(* IEC 61131-3 sources: repolevel_ST_code_completion/output/0127完整版本_带planner/repoeval_elevator/readful_result_no_provide, 4 files *)

(* ---- F_DetectCurrentFloor.st ---- *)
IF FloorSensor0 THEN
	F_DetectCurrentFloor := 0;
ELSIF FloorSensor1 THEN
	F_DetectCurrentFloor := 1;
ELSIF FloorSensor2 THEN
	F_DetectCurrentFloor := 2;
ELSIF FloorSensor3 THEN
	F_DetectCurrentFloor := 3;
ELSE
	F_DetectCurrentFloor := CurrentFloor;
END_IF;
RETURN;
END_FUNCTION

(* ---- F_UpdateDoorAnimation.st ---- *)
VAR
	nNewAni			:	DINT;		// 新的动画值
END_VAR

nNewAni := nCurrentAni;

// 开门动画（增加动画值）
IF bOpenDoor AND nNewAni < nMaxAni THEN
	nNewAni := nNewAni + 1;
END_IF

// 关门动画（减少动画值）
IF bCloseDoor AND nNewAni > 0 THEN
	nNewAni := nNewAni - 1;
END_IF

// 楼层呼叫动画（增加动画值）
IF bCallFloor AND nNewAni < nMaxAni THEN
	nNewAni := nNewAni + 1;
END_IF

// 保持动画值不变
IF NOT bCallFloor AND NOT bOpenDoor AND NOT bCloseDoor THEN
	nNewAni := nCurrentAni;
END_IF

F_UpdateDoorAnimation := nNewAni;
END_FUNCTION

(* ---- FB_ElevatorDoorController.st ---- *)
VAR
	fbDoorTimer			:	TON;		// 开门延时定时器
	fbCloseDoorTimer	:	TON;		// 关门延时定时器
	nState				:	INT;		// 状态机
	bEmergencyStop		:	BOOL;		// 紧急停止信号
END_VAR

CASE nState OF
	0: // 空闲状态
		bOpenDoor := FALSE;
		bCloseDoor := FALSE;
		bDoorOpen := FALSE;
		bDoorReady := TRUE;

		IF bArrivedAtTarget THEN
			nState := 1; // 开始开门流程
		END_IF

	1: // 开门延时
		bCloseDoor := FALSE;
		bDoorReady := FALSE;
		bOpenDoor := TRUE;
		fbDoorTimer(IN := TRUE, PT := T#2S);

		IF fbDoorTimer.Q THEN
			fbDoorTimer(IN := FALSE);
			nState := 2; // 门打开状态
		END_IF

	2: // 门打开状态
		bDoorOpen := TRUE;
		bOpenDoor := FALSE;

		IF NOT bArrivedAtTarget THEN
			nState := 3; // 开始关门流程
		END_IF

	3: // 关门延时
		bOpenDoor := FALSE;
		bDoorOpen := FALSE;
		bCloseDoor := TRUE;
		fbCloseDoorTimer(IN := TRUE, PT := T#2S);

		IF fbCloseDoorTimer.Q THEN
			fbCloseDoorTimer(IN := FALSE);
			nState := 4; // 检查门关闭状态
		END_IF

	4: // 检查门关闭状态
		bCloseDoor := FALSE;

		IF bDoorClosed THEN
			bDoorReady := TRUE;
			nState := 0; // 返回空闲状态
		END_IF

ELSE
	// 异常处理
	bOpenDoor := FALSE;
	bCloseDoor := FALSE;
	bDoorOpen := FALSE;
	bDoorReady := FALSE;
	nState := 0; // 返回空闲状态
END_CASE
END_FUNCTION_BLOCK

(* ---- FB_ElevatorMovement.st ---- *)
VAR
	i					:	INT;				// 循环变量
	bHasUpperRequest	:	BOOL;				// 有更高楼层请求
	bHasLowerRequest	:	BOOL;				// 有更低楼层请求
END_VAR

// 初始化状态变量
bHasUpperRequest := FALSE;
bHasLowerRequest := FALSE;

// 遍历目标楼层数组
FOR i := 0 TO 3 DO
	IF TargetFloors[i] THEN
		IF (i > CurrentFloor) AND bDoorReady THEN
			bHasUpperRequest := TRUE;
		ELSIF (i < CurrentFloor) AND bDoorReady THEN
			bHasLowerRequest := TRUE;
		END_IF;
	END_IF;
END_FOR

// 根据请求状态设置移动方向
IF bHasUpperRequest THEN
	bMovingUp := TRUE;
	bMovingDown := FALSE;
ELSIF bHasLowerRequest THEN
	bMovingDown := TRUE;
	bMovingUp := FALSE;
ELSE
	bMovingUp := FALSE;
	bMovingDown := FALSE;
END_IF

// 检查是否到达目标楼层
IF TargetFloors[CurrentFloor] THEN
	IF bDoorReady THEN
		bArrivedAtTarget := TRUE;
		TargetFloors[CurrentFloor] := FALSE; // 清除请求
		bMovingUp := FALSE;
		bMovingDown := FALSE;
	ELSE
		bArrivedAtTarget := FALSE;
	END_IF;
ELSE
	bArrivedAtTarget := FALSE;
END_IF
END_FUNCTION_BLOCK
